TYPE ST_HomeAbsEncoder :
STRUCT
	
	BlockOffsetPosition: 	LREAL; 
END_STRUCT
END_TYPE

(* stored: Version 1.1.0.1, ProductVersion 3.1.4024.3
   DUT ST_HomeAbsEncoder: Id {e468aa8e-7a1d-4d03-b1f9-f980cdfb5ba3} *)
